FUNCTION_BLOCK HeatCommand EXTENDS PLCopenCommand
VAR_INPUT
	TempSetPoint : REAL;
END_VAR

END_FUNCTION_BLOCK

(* stored: Version 1.1.0.1
   POU HeatCommand: Id {609cd9e9-f0c3-01ef-2b21-0fd9e152277f}, SpecialFunc None *)
